// TIA Portal V17 export
// export: Created 2023-12-22T15:07:58.5361564Z, ExportSetting WithDefaults, DisplayName Totally Integrated Automation Portal, DisplayVersion V17, DisplayName TIA Portal Openness, DisplayVersion V17, DisplayName TIA Portal Version Control Interface, DisplayVersion V17, DisplayName STEP 7 Professional, DisplayVersion V17, DisplayName STEP 7 Safety, DisplayVersion V17, DisplayName WinCC Advanced, DisplayVersion V17
ORGANIZATION_BLOCK "Main"   // OB1, LAD, ProgramCycle
TITLE = "Main Program Sweep (Cycle)"
{ S7_Optimized_Access := 'TRUE' }
VERSION : 0.1
// stored: AutoNumber true, IsIECCheckEnabled false, SetENOAutomatically false
   VAR_INPUT
      Initial_Call : Bool;   // Initial call of this OB
      Remanence : Bool;   // =True, if remanent data are available
   END_VAR
   VAR_TEMP   // added for the SCL form of the ladder/FBD networks
      _w1 : Bool;
   END_VAR
BEGIN

REGION Network 1
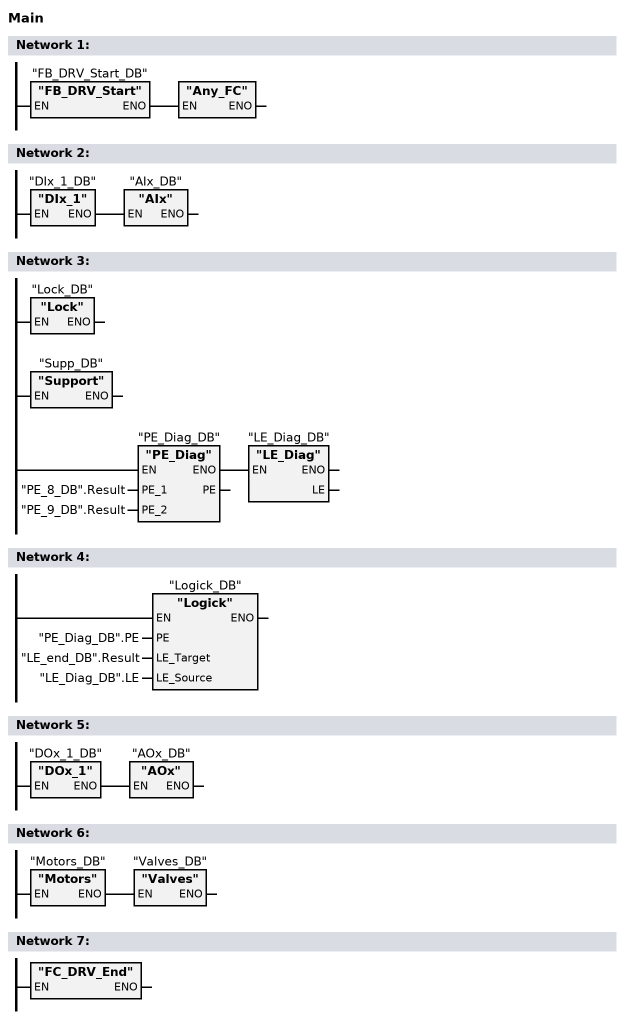
   RUNG wire#powerrail
      "FB_DRV_Start_DB"()
      "Any_FC"()
   END_RUNG
   // the same network as SCL:
   "FB_DRV_Start_DB"(ENO => #_w1);   // "FB_DRV_Start"
   IF #_w1 THEN "Any_FC"(); END_IF;
END_REGION

REGION Network 2
   RUNG wire#powerrail
      "DIx_1_DB"()
      "AIx_DB"()
   END_RUNG
   // the same network as SCL:
   "DIx_1_DB"(ENO => #_w1);   // "DIx_1"
   IF #_w1 THEN
       "AIx_DB"();   // "AIx"
   END_IF;
END_REGION

REGION Network 3
   RUNG wire#powerrail
      "Lock_DB"()
   END_RUNG
   RUNG wire#powerrail
      "Supp_DB"()
   END_RUNG
   RUNG wire#powerrail
      "PE_Diag_DB"(PE_1 := "PE_8_DB".Result, PE_2 := "PE_9_DB".Result, PE =>)
      "LE_Diag_DB"(LE =>)
   END_RUNG
   // the same network as SCL:
   "Lock_DB"();   // "Lock"
   "Supp_DB"();   // "Support"
   "PE_Diag_DB"(PE_1 := "PE_8_DB".Result, PE_2 := "PE_9_DB".Result, ENO => #_w1);   // "PE_Diag"
   IF #_w1 THEN
       "LE_Diag_DB"();   // "LE_Diag"
   END_IF;
END_REGION

REGION Network 4
   RUNG wire#powerrail
      "Logick_DB"(PE := "PE_Diag_DB".PE, LE_Target := "LE_end_DB".Result, LE_Source := "LE_Diag_DB".LE)
   END_RUNG
   // the same network as SCL:
   "Logick_DB"(PE := "PE_Diag_DB".PE, LE_Target := "LE_end_DB".Result, LE_Source := "LE_Diag_DB".LE);   // "Logick"
END_REGION

REGION Network 5
   RUNG wire#powerrail
      "DOx_1_DB"()
      "AOx_DB"()
   END_RUNG
   // the same network as SCL:
   "DOx_1_DB"(ENO => #_w1);   // "DOx_1"
   IF #_w1 THEN
       "AOx_DB"();   // "AOx"
   END_IF;
END_REGION

REGION Network 6
   RUNG wire#powerrail
      "Motors_DB"()
      "Valves_DB"()
   END_RUNG
   // the same network as SCL:
   "Motors_DB"(ENO => #_w1);   // "Motors"
   IF #_w1 THEN
       "Valves_DB"();   // "Valves"
   END_IF;
END_REGION

REGION Network 7
   RUNG wire#powerrail
      "FC_DRV_End"()
   END_RUNG
   // the same network as SCL:
   "FC_DRV_End"();
END_REGION
END_ORGANIZATION_BLOCK
